// Block: JB_PERS

DATA_BLOCK JB_PERS
VERSION : 0.1
   NON_RETAIN
   VAR
      PersistentValues : Struct
         Data : Struct
            WeldingSetUp : JB_WeldingSetUp;
            ClampEntryClosed : Bool;
            ClampExitClosed : Bool;
         END_STRUCT;
         Torch : Struct
            MeasureTorchHolder : LReal;
            InhibitWeld_Pos : LReal;
            InhibitWeld_Window : LReal;
            Parking_Pos : LReal;
            WeldingUseLocalData : Bool;
            Cycle_HighSpeed : LReal;
            Cycle_LowSpeed : LReal;
         END_STRUCT;
         TorchAx : Positioning_DOL_Machine_Par;
         TorchAx_Pers : Positioning_DOL_Machine_Pers_Data;
         TorchEnc : PosFbk_RTN;
         PinchRoll_Feed : SpeedMachine_Par;
         Aspiratore_TimeOff : Time;
      END_STRUCT;
   END_VAR

BEGIN
   // No initialization required
END_DATA_BLOCK
